// TIA Portal V21 export
VAR_GLOBAL   // PLC tag table "Cabinet_Management"
   M_Power_cabinet AT %M2.0 : Bool;
   M_Power_L1 AT %M3.0 : Bool;
   M_Power_L2 AT %M3.1 : Bool;
   M_Power_L3 AT %M3.2 : Bool;
   M_Power_L4 AT %M3.3 : Bool;
   M_Power_L5 AT %M3.4 : Bool;
   M_Power_L6 AT %M3.5 : Bool;
   M_Buzzer AT %M4.0 : Bool;
   M_NF_Cabinet_fault AT %M5.0 : Bool;
   M_Cabinet_fault AT %M5.1 : Bool;
   M_Rearm_Power_Cabinet AT %M6.0 : Bool;
   M_Reset_safety_Z1 AT %M7.0 : Bool;
   M_Reset_safety_Z2 AT %M7.1 : Bool;
   M_Reset_safety_Z3 AT %M7.2 : Bool;
   M_Reset_safety_Z4 AT %M7.3 : Bool;
   M_Reset_safety_Z5 AT %M7.4 : Bool;
   M_Reset_safety_Z6 AT %M7.5 : Bool;
   M_Reset_safety_Z7 AT %M7.6 : Bool;
   M_Reset_safety_Z8 AT %M7.7 : Bool;
   M_Facility_OK AT %M6.7 : Bool;   // Conveyors status OK
END_VAR
